// TIA Portal V20 export
TYPE "LKinCtrl_typeKinematicsZoneDefinition"
   STRUCT
      coordinateSystem : DInt;   // 0:FCS, 1:TCS
      frame : "LKinCtrl_typeFrame";   // shifting of the zone zero point in relation to the reference system
      geometryType : DInt;   // 0:Cuboid, 1:Sphere, 2:Cylinder
      geometryParameter : Array[1..3] of LReal;   // geometry parameter depending on geometry type
   END_STRUCT;
END_TYPE
